PROGRAM SIMULATION
VAR
	TON_0: TON;
	TON_1: TON;
	TON_2: TON;
	TON_3: TON;
	TON_4: TON;
	bPAL_M882A			:BOOL:=TRUE;
	TON_5: TON;
	TON_6: TON;
	TON_7: TON;
	TON_8: TON;
	
	rMixerAngle			:REAL;
	iRevolutions		:INT;
	tonMixerRPM			:TON;
	fbScaleMixerRev		:FB_Scale;
END_VAR


VAR PERSISTENT
	TIME_5: TIME;
	TIME_6: TIME;
END_VAR
VAR // added by the converter: edge detectors and wires of the graphical bodies
    _w1, _w2, _w3 : BOOL;
END_VAR

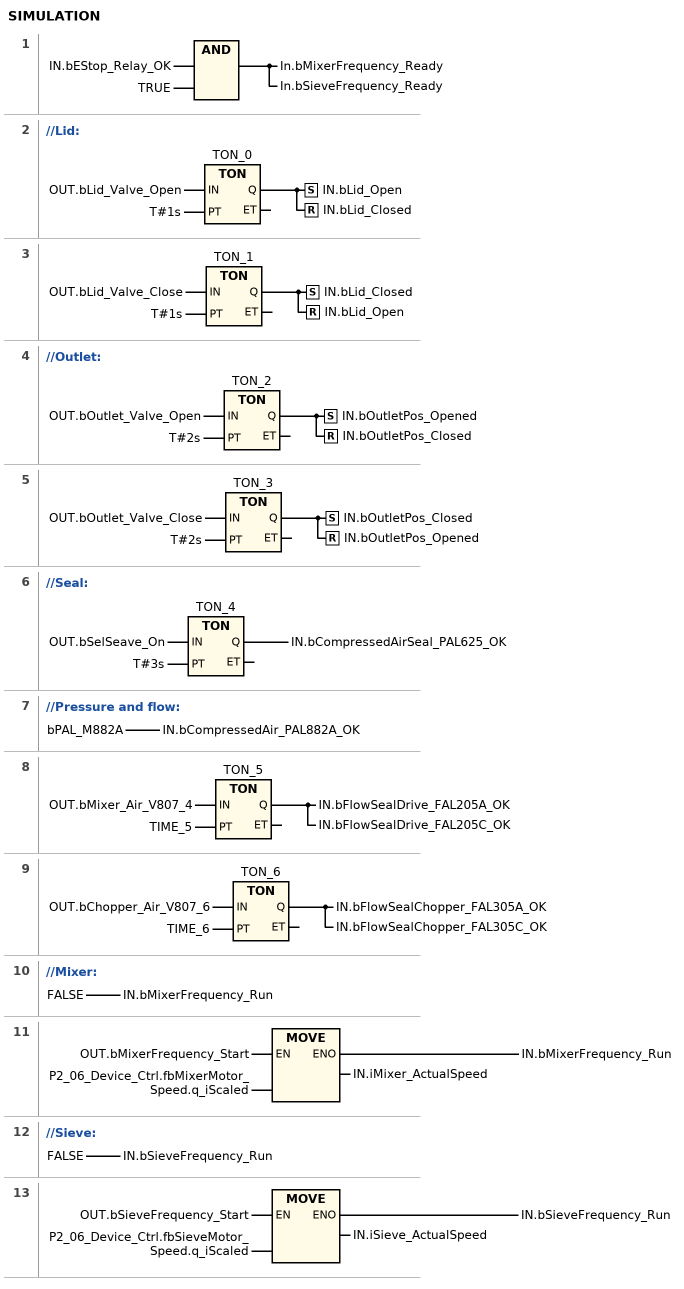
// NETWORK 1
_w1 := IN.bEStop_Relay_OK AND TRUE;
In.bMixerFrequency_Ready := _w1;
In.bSieveFrequency_Ready := _w1;

// NETWORK 2
// label: //Lid
TON_0(IN := OUT.bLid_Valve_Open, PT := T#1s); // TON
IN.bLid_Open S= TON_0.Q;
IN.bLid_Closed R= TON_0.Q;

// NETWORK 3
TON_1(IN := OUT.bLid_Valve_Close, PT := T#1s); // TON
IN.bLid_Closed S= TON_1.Q;
IN.bLid_Open R= TON_1.Q;

// NETWORK 4
// label: //Outlet
TON_2(IN := OUT.bOutlet_Valve_Open, PT := T#2s); // TON
IN.bOutletPos_Opened S= TON_2.Q;
IN.bOutletPos_Closed R= TON_2.Q;

// NETWORK 5
TON_3(IN := OUT.bOutlet_Valve_Close, PT := T#2s); // TON
IN.bOutletPos_Closed S= TON_3.Q;
IN.bOutletPos_Opened R= TON_3.Q;

// NETWORK 6
// label: //Seal
TON_4(IN := OUT.bSelSeave_On, PT := T#3s); // TON
IN.bCompressedAirSeal_PAL625_OK := TON_4.Q;

// NETWORK 7
// label: //Pressure and flow
IN.bCompressedAir_PAL882A_OK := bPAL_M882A;

// NETWORK 8
TON_5(IN := OUT.bMixer_Air_V807_4, PT := TIME_5); // TON
IN.bFlowSealDrive_FAL205A_OK := TON_5.Q;
IN.bFlowSealDrive_FAL205C_OK := TON_5.Q;

// NETWORK 9
TON_6(IN := OUT.bChopper_Air_V807_6, PT := TIME_6); // TON
IN.bFlowSealChopper_FAL305A_OK := TON_6.Q;
IN.bFlowSealChopper_FAL305C_OK := TON_6.Q;

// NETWORK 10
// label: //Mixer
IN.bMixerFrequency_Run := FALSE;

// NETWORK 11
_w2 := OUT.bMixerFrequency_Start;
IF _w2 THEN IN.iMixer_ActualSpeed := P2_06_Device_Ctrl.fbMixerMotor_Speed.q_iScaled; END_IF
IN.bMixerFrequency_Run := _w2;

// NETWORK 12
// label: //Sieve
IN.bSieveFrequency_Run := FALSE;

// NETWORK 13
_w3 := OUT.bSieveFrequency_Start;
IF _w3 THEN IN.iSieve_ActualSpeed := P2_06_Device_Ctrl.fbSieveMotor_Speed.q_iScaled; END_IF
IN.bSieveFrequency_Run := _w3;

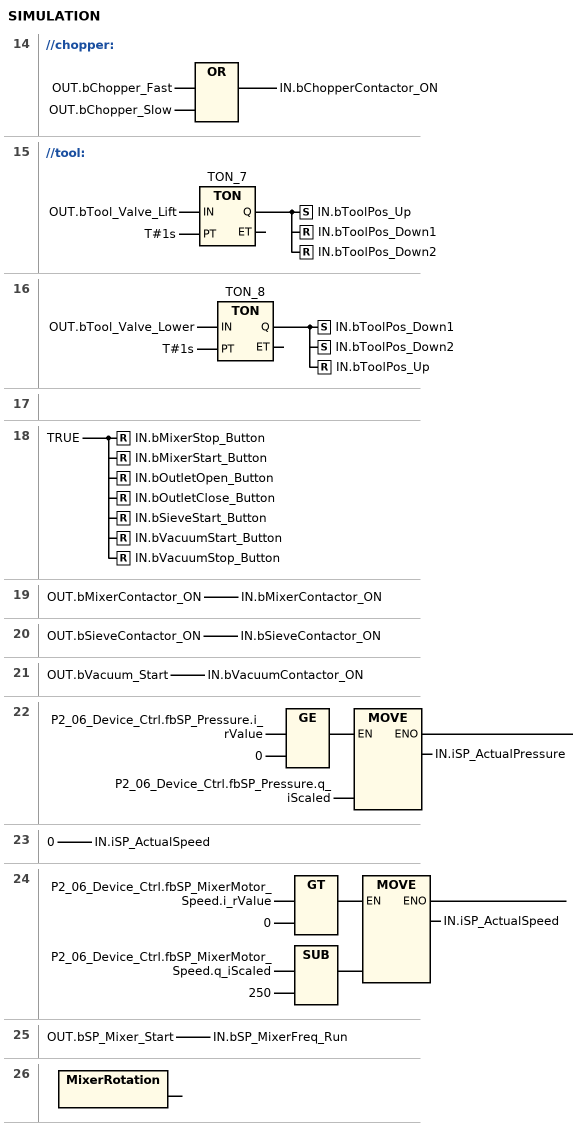
// NETWORK 14
// label: //chopper
IN.bChopperContactor_ON := OUT.bChopper_Fast OR OUT.bChopper_Slow;

// NETWORK 15
// label: //tool
TON_7(IN := OUT.bTool_Valve_Lift, PT := T#1s); // TON
IN.bToolPos_Up S= TON_7.Q;
IN.bToolPos_Down1 R= TON_7.Q;
IN.bToolPos_Down2 R= TON_7.Q;

// NETWORK 16
TON_8(IN := OUT.bTool_Valve_Lower, PT := T#1s); // TON
IN.bToolPos_Down1 S= TON_8.Q;
IN.bToolPos_Down2 S= TON_8.Q;
IN.bToolPos_Up R= TON_8.Q;

// NETWORK 17

// NETWORK 18
IN.bMixerStop_Button R= TRUE;
IN.bMixerStart_Button R= TRUE;
IN.bOutletOpen_Button R= TRUE;
IN.bOutletClose_Button R= TRUE;
IN.bSieveStart_Button R= TRUE;
IN.bVacuumStart_Button R= TRUE;
IN.bVacuumStop_Button R= TRUE;

// NETWORK 19
IN.bMixerContactor_ON := OUT.bMixerContactor_ON;

// NETWORK 20
IN.bSieveContactor_ON := OUT.bSieveContactor_ON;

// NETWORK 21
IN.bVacuumContactor_ON := OUT.bVacuum_Start;

// NETWORK 22
IF P2_06_Device_Ctrl.fbSP_Pressure.i_rValue >= 0 THEN
    IN.iSP_ActualPressure := P2_06_Device_Ctrl.fbSP_Pressure.q_iScaled;
END_IF

// NETWORK 23
IN.iSP_ActualSpeed := 0;

// NETWORK 24
IF P2_06_Device_Ctrl.fbSP_MixerMotor_Speed.i_rValue > 0 THEN
    IN.iSP_ActualSpeed := P2_06_Device_Ctrl.fbSP_MixerMotor_Speed.q_iScaled - 250;
END_IF

// NETWORK 25
IN.bSP_MixerFreq_Run := OUT.bSP_Mixer_Start;

// NETWORK 26
MixerRotation();

ACTION MixerRotation:

tonMixerRPM(IN:=P2_06_Device_Ctrl.fbMixerMotor_Speed.i_rValue<>0 AND OUT.bMixerFrequency_Start AND NOT tonMixerRPM.Q ,
			PT:=TO_TIME(P2_06_Device_Ctrl.fbMixerMotor_Speed.i_rValue/60*1000));

IF tonMixerRPM.Q THEN
	iRevolutions:=iRevolutions+1;
END_IF

IF iRevolutions > 32000 THEN
	iRevolutions:=0;
END_IF
IF TO_REAL(tonMixerRPM.PT) <> 0 THEN
	fbScaleMixerRev(i_rValue:=TO_REAL(tonMixerRPM.ET),
					i_rRawData_Low:=0,
					i_rRawData_High:=TO_REAL(tonMixerRPM.PT),
					i_rScaled_Low:=0,
					i_rScaled_High:=360,
					i_rOffset:=0,
					q_rScaled=>rMixerAngle);
END_IF	
IF rMixerAngle > 100 AND rMixerAngle < 150 THEN
	IN.bMixerTool_InPos:=TRUE;
ELSE
	IN.bMixerTool_InPos:=FALSE;
END_IF
END_ACTION

END_PROGRAM

(* stored: Version 1.1.0.1, ProductVersion 3.1.4024.12
   POU SIMULATION: Id {f5820b0f-8b6c-4003-97a5-49d5e27f7c5f}, SpecialFunc None
   Action MixerRotation: Id {dc2c7f23-07e4-4a87-be2c-d4e607a6945e} *)
